FUNCTION_BLOCK EL1202
VAR
	_io : EL1xx2_Data;
	{attribute addProperty Name "WcState"}
	_wcState : WcStateInputToggle;
	{attribute addProperty Name "Info data"}
	_infoData : InfoDataBase;
END_VAR

PROPERTY IO : REFERENCE TO EL1xx2_Data
GET
IO REF= _io;
END_GET
END_PROPERTY

PROPERTY WcState : REFERENCE TO WcStateInputToggle
GET
WcState REF= _wcState;
END_GET
END_PROPERTY

END_FUNCTION_BLOCK

(* stored: Version 1.1.0.1, ProductVersion 3.1.4024.9
   POU EL1202: Id {7cff48be-eef0-0bc8-3497-26abbac9a20b}, SpecialFunc None
   Property IO: Id {8ae5c645-4e1e-06f9-0957-82079b632915}
   Get Get: Id {e52ae162-60f0-0c56-0a6e-9b3b45f49146}
   Property WcState: Id {6274a6e4-718e-06df-1ddf-13827ae02b4f}
   Get Get: Id {1b617e10-8ae2-0a36-3f43-69f2e446d2ef} *)
